Staubli VAL3: _resetAllPallet.pjx

--- _resetAllPallet.pjx ---
Parameters version=s7.2.1 stackSize=5000 millimeterUnit=true
Program file=resetAllPallet.pgx
Program file=start.pgx
Program file=stop.pgx
Data file=_resetAllPallet.dtx
Library alias=pallet path=Disk://trajectory/PALLET/PALLET.pjx
Library alias=OnEvent path=Disk://OnEvent/OnEvent.pjx
Library alias=saveData path=Disk://saveData/saveData.pjx

--- _resetAllPallet.dtx ---
string sPalletName
mdesc nom_speed = {rmax=9999, blend=off}

--- start.pgx ---
public program start()
begin
  call resetAllPallet()
end

--- getPalletList.pgx ---
program getPalletList()
begin
  //
  // INIT
  //
  libList(saveData:sPathTraj+"PALLET",sPalletName)
end

--- resetAllPallet.pgx ---
program resetAllPallet()
  local num i
  local string l_sPalletName
begin
  // resetALL
  call pallet:reset()
  // call the onEvent procedure
  call OnEvent:OnCycleEvent(16)
end
